Omron CX-Programmer project NewProject (CX-Programmer 9.70)

# PLC NewPLC1: CP1E E20

## Global symbols (name address type ; comment)
0.01 BOOL  ; start

## Program NewProgram1 (cyclic task 0)

### Section Section1

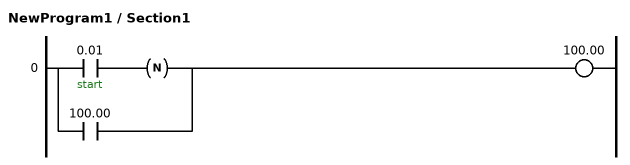
; rung 0
LD 0.01  ; start
DOWN(522)
OR 100.00
OUT 100.00

### Section END
; rung 0
END(001)